Fanuc KAREL source: ks00052.KL

-- PROVISIONAL review KL for V1013-1; original PC SHA256 f52ba2a2242c3406bf7b1895764617cd0f0d8df1ca6621ca0ed8eebba3a4338d
-- Incomplete behavior may be omitted. Consult companion uncertainty JSON. Do not deploy.
PROGRAM KS00052
%NOLOCKGROUP
BEGIN
  -- UNRESOLVED_PC offsets 5-13; opcodes 3F,75
  -- UNRESOLVED_PC offsets 18-27; opcodes 3F,75
  -- UNRESOLVED_PC offsets 32-46; opcodes 22,22,1E
  -- UNRESOLVED_PC offsets 51-55; opcodes 7F
END KS00052
